Universal Robots PolyScope program: roof_b.urp

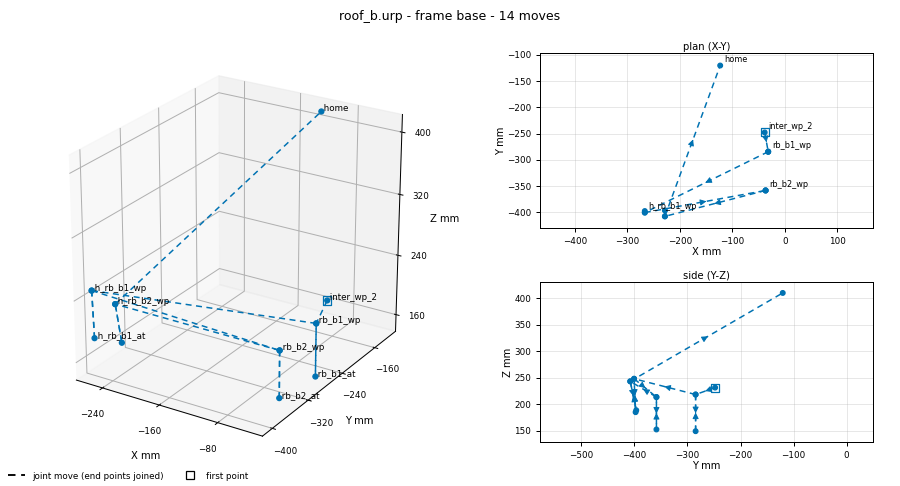
[picture p0: tool path of roof_b.urp in frame base, 14 of 14 moves have a stored position in this frame; points joined in program order, loops and branches not executed]
Program roof_b (installation=default directory=/programs/Session 1 createdIn=5.3.1.64192 lastSavedIn=5.3.1.64192 robotSerialNumber=20195300365)
Calibrated DH parameters: a=[-0.000093, -0.190649, -0.212673, 0.000091, -0.000205, 0]; d=[0.151591, 44.061648, -42.488068, -1.442789, 0.085322, 0.091911]; alpha=[1.570082, -0.003447, 0.007513, 1.572293, -1.571904, 0]; deltaTheta=[0, -0.672656, 0.728185, -0.055522, 0.000005, 0]
Robot Program (runOnlyOnce=true)
  URCap Gripper Activate (Robotiq_Grippers, Robotiq Inc.) dataModel(ResetAndActivateKey=false)
  URCap Gripper (Robotiq_Grippers, Robotiq Inc.) dataModel(position=50.0, force=100.0, speed=100.0, positionInDouble=50.0, forceInDouble=100.0, speedInDouble=100.0, slaveIds=[9], blocking=true)
  MoveJ speed 60 deg/s, acceleration 80 deg/s^2 (useActiveTCP=true) feature=Base
    Waypoint inter_wp_2: TCP in base x=-38.107 y=-247.898 z=231.572 mm, rx=2.241 ry=2.1798 rz=0.019 rad; joints [-68.076, -72.135, -124.793, -72.457, 91.361, -246.109] deg
  Folder Roof_B
    MoveJ speed 60 deg/s, acceleration 80 deg/s^2 (useActiveTCP=true) feature=Base
      Waypoint rb_b1_wp: TCP in base x=-31.427 y=-284.614 z=218.562 mm, rx=2.2451 ry=2.1882 rz=-0.0171 rad; joints [-69.272, -83.632, -119.946, -65.773, 89.911, -247.396] deg
      Waypoint rb_b1_at: TCP in base x=-31.436 y=-284.602 z=149.414 mm, rx=2.2452 ry=2.1882 rz=-0.017 rad; joints [-69.305, -95.054, -131.489, -42.815, 89.791, -247.308] deg
      URCap Gripper (Robotiq_Grippers, Robotiq Inc.) dataModel(position=100.0, force=100.0, speed=100.0, positionInDouble=100.0, forceInDouble=100.0, speedInDouble=100.0, slaveIds=[9], blocking=true)
      Waypoint rb_b1_wp: TCP in base x=-31.427 y=-284.614 z=218.562 mm, rx=2.2451 ry=2.1882 rz=-0.0171 rad; joints [-69.272, -83.632, -119.946, -65.773, 89.911, -247.396] deg
      Waypoint h_rb_b1_wp: TCP in base x=-266.628 y=-400.606 z=248.259 mm, rx=-2.9221 ry=0.0608 rz=-0.0496 rad; joints [-107.509, -142.729, -21.88, -117.881, 88.571, -195.052] deg
      Waypoint h_rb_b1_at: TCP in base x=-266.631 y=-397.735 z=185.295 mm, rx=-2.9221 ry=0.0608 rz=-0.0498 rad; joints [-107.672, -139.156, -45.769, -97.57, 88.599, -195.057] deg
      URCap Gripper (Robotiq_Grippers, Robotiq Inc.) dataModel(position=50.0, force=100.0, speed=100.0, positionInDouble=50.0, forceInDouble=100.0, speedInDouble=100.0, slaveIds=[9], blocking=true)
      Waypoint h_rb_b1_wp: TCP in base x=-266.628 y=-400.606 z=248.259 mm, rx=-2.9221 ry=0.0608 rz=-0.0496 rad; joints [-107.509, -142.729, -21.88, -117.881, 88.571, -195.052] deg
    MoveJ speed 60 deg/s, acceleration 80 deg/s^2 (useActiveTCP=true) feature=Base
      Waypoint rb_b2_wp: TCP in base x=-36.381 y=-358.469 z=213.765 mm, rx=-2.2634 ry=-2.1742 rz=-0.0315 rad; joints [-74.964, -103.256, -99.679, -67.697, 91.219, -252.317] deg
      Waypoint rb_b2_at: TCP in base x=-36.369 y=-358.47 z=152.678 mm, rx=-2.2633 ry=-2.1743 rz=-0.0315 rad; joints [-74.985, -110.842, -108.306, -51.483, 91.149, -252.255] deg
      URCap Gripper (Robotiq_Grippers, Robotiq Inc.) dataModel(position=100.0, force=100.0, speed=100.0, positionInDouble=100.0, forceInDouble=100.0, speedInDouble=100.0, slaveIds=[9], blocking=true)
      Waypoint rb_b2_wp: TCP in base x=-36.381 y=-358.469 z=213.765 mm, rx=-2.2634 ry=-2.1742 rz=-0.0315 rad; joints [-74.964, -103.256, -99.679, -67.697, 91.219, -252.317] deg
      Waypoint h_rb_b2_wp: TCP in base x=-228.341 y=-407.823 z=243.4 mm, rx=-2.9484 ry=0.091 rz=-0.0234 rad; joints [-102.754, -134.315, -39.474, -107.104, 89.06, -189.115] deg
      Waypoint h_rb_b2_at: TCP in base x=-228.326 y=-396.503 z=188.908 mm, rx=-2.9484 ry=0.091 rz=-0.0233 rad; joints [-103.117, -131.694, -58.874, -90.32, 89.017, -189.341] deg
      URCap Gripper (Robotiq_Grippers, Robotiq Inc.) dataModel(position=50.0, force=100.0, speed=100.0, positionInDouble=50.0, forceInDouble=100.0, speedInDouble=100.0, slaveIds=[9], blocking=true)
      Waypoint h_rb_b2_wp: TCP in base x=-228.341 y=-407.823 z=243.4 mm, rx=-2.9484 ry=0.091 rz=-0.0234 rad; joints [-102.754, -134.315, -39.474, -107.104, 89.06, -189.115] deg
  MoveJ speed 60 deg/s, acceleration 80 deg/s^2 (useActiveTCP=true) feature=Base
    Waypoint home: TCP in base x=-122.926 y=-120.377 z=410.038 mm, rx=2.273 ry=2.1657 rz=-0.0264 rad; joints [-85.876, -57.16, -80.452, -131.626, 89.649, -263.131] deg
